{attribute 'GeneratedUsingTerminal: EL6652-0000-0017'}
{attribute addProperty BoxType "EL6652-0000-0017"}
{attribute addProperty Id "InfoDataAT %I*InfoData_90184F0C16"}
{attribute addProperty CRC "554310285"}
{attribute addProperty Size "16"}
TYPE EL6652_210A1A8D EXTENDS EtcSlaveTerminalBase_947E5A46 :
STRUCT
	{attribute addProperty Name "InfoData"}
	InfoData : InfoData_90184F0C;
END_STRUCT
END_TYPE

(* stored: Version 1.2.0.0, ProductVersion 3.1.4024.9
   DUT EL6652_210A1A8D: Id {2a881c74-14e0-4cc4-a4eb-83cf63293847} *)
